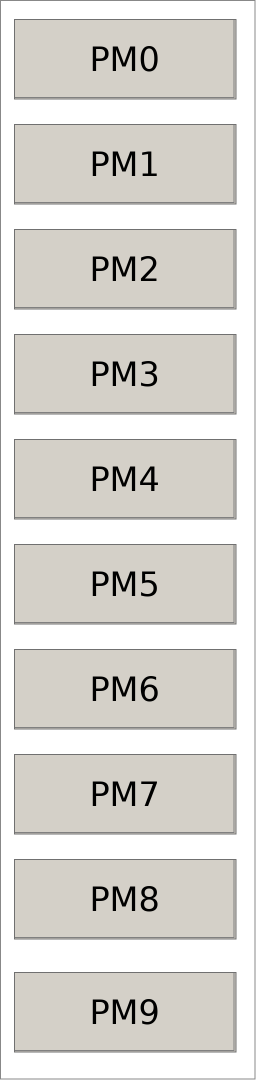
VISUALIZATION PMList  // 256x1080
    Button (1413,1160 244x110), "ReM0"
        OnMouseDown: execute { G_HMI.iMainFrame  := 0; }
    Button (14,19 222x80), "PM0", colour toggle: G_HMI.iPM =0
        p573394764: 16#FF00FF00
        OnMouseDown: execute { G_HMI.iPM  := 0; G_HMI.iMainFrame	:= 1; }
    Button (14,124 222x80), "PM1", colour toggle: G_HMI.iPM =1
        p573394764: 16#FF00FF00
        OnMouseDown: execute { G_HMI.iPM  := 1; G_HMI.iMainFrame	:= 1; }
    Button (14,229 222x80), "PM2", colour toggle: G_HMI.iPM =2
        p573394764: 16#FF00FF00
        OnMouseDown: execute { G_HMI.iPM  := 2; G_HMI.iMainFrame	:= 1; }
    Button (14,334 222x80), "PM3", colour toggle: G_HMI.iPM =3
        p573394764: 16#FF00FF00
        OnMouseDown: execute { G_HMI.iPM  := 3; G_HMI.iMainFrame	:= 1; }
    Button (14,439 222x80), "PM4", colour toggle: G_HMI.iPM =4
        p573394764: 16#FF00FF00
        OnMouseDown: execute { G_HMI.iPM  := 4; G_HMI.iMainFrame	:= 1; }
    Button (14,544 222x80), "PM5", colour toggle: G_HMI.iPM =5
        p573394764: 16#FF00FF00
        OnMouseDown: execute { G_HMI.iPM  := 5; G_HMI.iMainFrame	:= 1; }
    Button (14,649 222x80), "PM6", colour toggle: G_HMI.iReM =6
        p573394764: 16#FF00FF00
        OnMouseDown: execute { G_HMI.iPM  := 6; G_HMI.iMainFrame	:= 1; }
    Button (14,754 222x80), "PM7", colour toggle: G_HMI.iReM =7
        p573394764: 16#FF00FF00
        OnMouseDown: execute { G_HMI.iPM  := 7; G_HMI.iMainFrame	:= 1; }
    Button (14,859 222x80), "PM8", colour toggle: G_HMI.iReM =8
        p573394764: 16#FF00FF00
        OnMouseDown: execute { G_HMI.iPM  := 8; G_HMI.iMainFrame	:= 1; }
    Button (14,972 222x80), "PM9", colour toggle: G_HMI.iReM =9
        p573394764: 16#FF00FF00
        OnMouseDown: execute { G_HMI.iPM  := 9; G_HMI.iMainFrame	:= 1; }
END_VISUALIZATION

(* stored: Version 1.1.0.1, ProductVersion 3.1.4024.12
   Visu PMList: Id {53d37355-9046-4a04-815f-2ac247117e3a} *)
